{attribute 'linkalways'} 
{attribute 'no_explicit_call' := 'This FB is a CLASS and must be accessed using methods or properties'}
{attribute 'enable_dynamic_creation'}
FUNCTION_BLOCK _Array0to3OfTcVnPoint2_REAL EXTENDS ArrayDatatypeBase
VAR CONSTANT
	lBound : DINT := 0;
	uBound : DINT := 3;
END_VAR
VAR
	localData : ARRAY [lBound..uBound] OF TcVnPoint2_REAL;
	activeData : REFERENCE TO ARRAY [lBound..uBound] OF TcVnPoint2_REAL REF= localData;
	elements : ARRAY [lBound..uBound] OF _TcVnPoint2_REAL;
	baseType : _TcVnPoint2_REAL;
END_VAR

PROPERTY PUBLIC Address : PVOID
GET
Address := ADR(activeData);
END_GET
END_PROPERTY

PROPERTY PUBLIC BaseDatatype : I_Datatype
GET
BaseDatatype := baseType;
END_GET
END_PROPERTY

METHOD PUBLIC ClearReference
VAR_INPUT
END_VAR
activeData REF= localData;
SetElementReference();
END_METHOD

METHOD PUBLIC Clone : I_Datatype
VAR
    pClone : POINTER TO _Array0to3OfTcVnPoint2_REAL;
END_VAR
pClone := __NEW(_Array0to3OfTcVnPoint2_REAL());
pClone^.Value := Value;
Clone := pClone^;
END_METHOD

METHOD FB_init : BOOL
VAR_INPUT
	bInitRetains : BOOL; // if TRUE, the retain variables are initialized (warm start / cold start)
	bInCopyCode : BOOL;  // if TRUE, the instance afterwards gets moved into the copy code (online change)
END_VAR
SetElementReference();
END_METHOD

METHOD PUBLIC GetElementAsDatatypeByIndex : I_Datatype
VAR_INPUT
	Index : DINT;
END_VAR
GetElementAsDatatypeByIndex := elements[Index];
END_METHOD

METHOD PUBLIC GetElementByIndex : REFERENCE TO _TcVnPoint2_REAL;
VAR_INPUT
	Index : DINT;
END_VAR
GetElementByIndex REF= elements[Index];
END_METHOD

PROPERTY PUBLIC LowerBound : DINT
GET
LowerBound := lBound;
END_GET
END_PROPERTY

METHOD PUBLIC MakeReferenceTo
VAR_INPUT
	ReferenceTarget : REFERENCE TO ARRAY [lBound..uBound] OF TcVnPoint2_REAL;
END_VAR
activeData REF= ReferenceTarget;
SetElementReference();
END_METHOD

METHOD PROTECTED OnSerializeArrayValues
VAR_INPUT
	Serializer : I_Serializer;
END_VAR
VAR
	i : DINT;
END_VAR
FOR i := lBound TO uBound DO
	elements[i].SerializeWith(Serializer);
END_FOR
END_METHOD

METHOD PROTECTED SetElementReference
VAR_INPUT
END_VAR
VAR
	i : DINT;
END_VAR
FOR i := lBound TO uBound DO
	elements[i].MakeReferenceTo(activeData[i]);
END_FOR
END_METHOD

PROPERTY PUBLIC Size : UDINT
GET
Size := SIZEOF(activeData);
END_GET
END_PROPERTY

METHOD PROTECTED TryDeserializeArrayValues : BOOL
VAR_INPUT
	Deserializer : I_Deserializer;
	Feedback : I_DeserializerFeedback;
END_VAR
VAR
	enumerator : I_DeserializerArrayForwardEnumerator;
	i : DINT;
END_VAR
enumerator := Deserializer.GetArrayEnumerator();
i := lBound;

WHILE enumerator.MoveNext() AND i <= uBound DO
	
	IF NOT elements[i].TryDeserializeFrom(enumerator.Current, Feedback) THEN
		EXIT;
	END_IF
	i := i + 1;

END_WHILE
enumerator.Dispose();
END_METHOD

METHOD TryMakeReferenceTo : BOOL
VAR_INPUT
	Target : I_Datatype;
END_VAR
VAR
	targetAsArray : I_ArrayDatatype;
	pTargetData : POINTER TO ARRAY [lBound..uBound] OF TcVnPoint2_REAL;
END_VAR
IF NOT Target.TryResolveAsArrayDatatype(targetAsArray) THEN
	RETURN;
END_IF

IF NOT (targetAsArray.Identifier = Identifier) THEN
	RETURN;
END_IF

pTargetData := Target.Address;
activeData REF= pTargetData^;
SetElementReference();
TryMakeReferenceTo := TRUE;
END_METHOD

PROPERTY PUBLIC UpperBound : DINT
GET
UpperBound := ubound;
END_GET
END_PROPERTY

PROPERTY PUBLIC Value : REFERENCE TO ARRAY [lBound..uBound] OF TcVnPoint2_REAL;
GET
Value ref= activeData;
END_GET
END_PROPERTY

END_FUNCTION_BLOCK

(* stored: Version 1.1.0.1, ProductVersion 3.1.4024.13
   POU _Array0to3OfTcVnPoint2_REAL: Id {703dfda6-c000-0f18-0d15-fc78879731cb}, SpecialFunc None
   Folder Core: Id {8fe21143-6790-0574-382a-1b5e1e3c06c0}
   Folder Constructor: Id {7ffd1a43-eecb-0ba3-081f-05b47356ba16}
   Folder Protected: Id {6593853e-75db-0312-0677-535ed3e1f2a8}
   Folder Customize: Id {230175c2-c49e-06e8-1001-c65a63338617}
   Property Address: Id {686fab7d-1ad4-0dc9-10f8-9b0227c61cba}
   Get Get: Id {56185003-5d85-0553-18ec-961304a9d326}
   Property BaseDatatype: Id {409122be-66b0-0245-0cde-82a885f75a6e}
   Get Get: Id {f42a9223-2702-0ab7-20b4-880f7eec66ec}
   Method ClearReference: Id {0d5a6d36-8edc-0122-1ba7-719c9a6d49ef}
   Method Clone: Id {8a009272-f976-0cdd-2a3d-7d964d268348}
   Method FB_init: Id {3bdf68c9-9ee3-0d81-1f3e-617fc65d19db}
   Method GetElementAsDatatypeByIndex: Id {958db28e-477d-0790-2213-832e1a7aa255}
   Method GetElementByIndex: Id {70cde067-20ab-0f3d-065c-b17db526bc99}
   Property LowerBound: Id {4649e062-9b0d-0321-09d2-07c7cdc1aec1}
   Get Get: Id {3fc1e2e5-304a-0395-1017-54def72d6834}
   Method MakeReferenceTo: Id {6f8f89f7-58a5-026e-2502-4abf557147f5}
   Method OnSerializeArrayValues: Id {d94d01a2-5e8d-0b5e-1299-d0635c476e63}
   Method SetElementReference: Id {7257bd73-fad2-0b94-3e4d-6dbbc02f5a27}
   Property Size: Id {74af6369-28dd-0bea-03cf-5b76b4995852}
   Get Get: Id {c75788c7-88c4-0cde-1f86-2e2bf81ee247}
   Method TryDeserializeArrayValues: Id {cfc66731-4a4a-08ab-0dfe-86cab639b4b1}
   Method TryMakeReferenceTo: Id {6d3af753-dba3-0258-3892-da016817c32f}
   Property UpperBound: Id {33bd46a9-24c8-07ce-3eb9-94bfc1171dae}
   Get Get: Id {72fc7a28-8227-0461-22a9-91270a4653d6}
   Property Value: Id {c7df7f1a-451f-0174-29a5-9e01fde4c3b7}
   Get Get: Id {bbac7f95-fe3d-02eb-35db-ecb80dcc5c4a} *)
